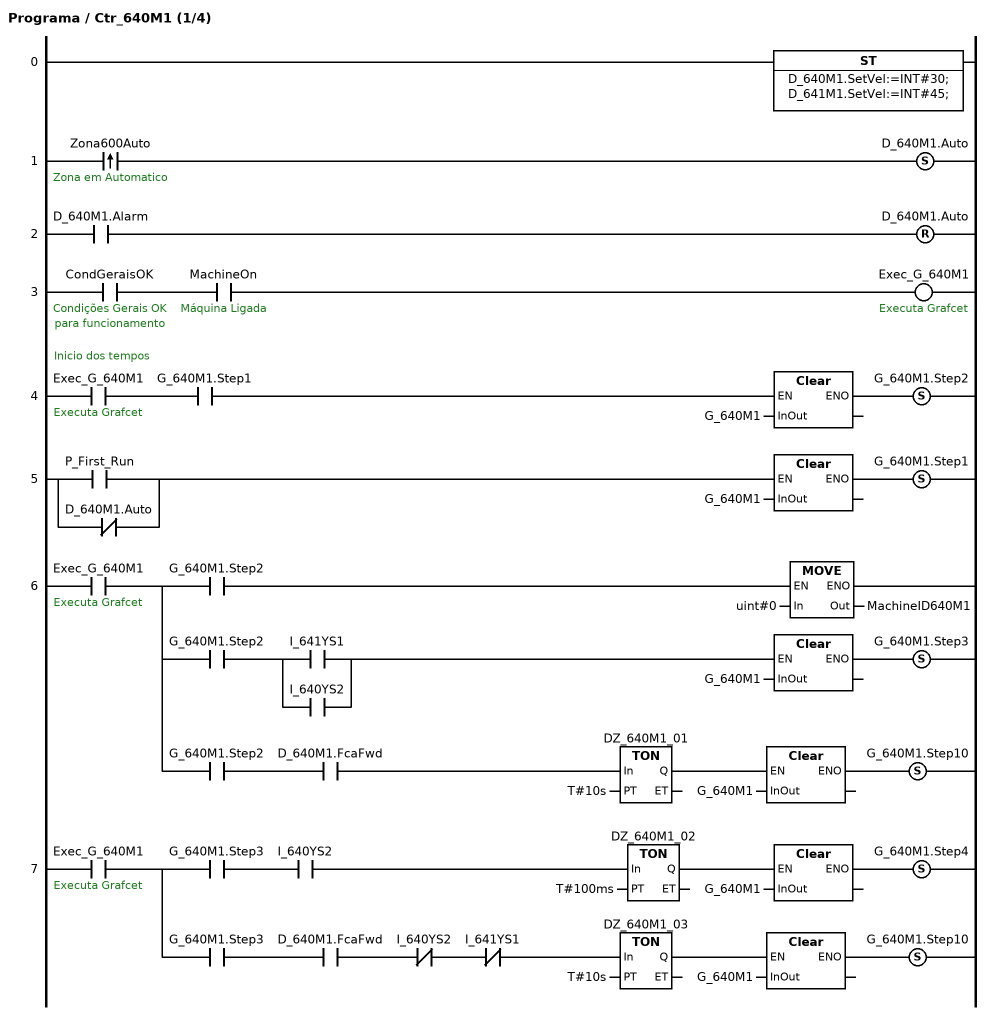
(* [picture p144: Programa / Ctr_640M1, rungs 0-7] *)
(* Rung 0 *)
D_640M1.SetVel:=INT#30;
D_641M1.SetVel:=INT#45;
(* Rung 1 *)
_e291(CLK := Zona600Auto);
IF _e291.Q THEN D_640M1.Auto := TRUE; END_IF;
(* Rung 2 *)
IF D_640M1.Alarm THEN D_640M1.Auto := FALSE; END_IF;
(* Rung 3 *)
Exec_G_640M1 := CondGeraisOK AND MachineOn;
(* Rung 4: Inicio dos tempos *)
_p292 := Exec_G_640M1 AND G_640M1.Step1;
IF _p292 THEN
    Clear(InOut := G_640M1);
    G_640M1.Step2 := TRUE;
END_IF;
(* Rung 5 *)
IF P_First_Run OR NOT D_640M1.Auto THEN
    Clear(InOut := G_640M1);
    G_640M1.Step1 := TRUE;
END_IF;
(* Rung 6 *)
IF Exec_G_640M1 AND G_640M1.Step2 THEN MachineID640M1 := uint#0; END_IF;
_p293 := Exec_G_640M1 AND G_640M1.Step2 AND (I_641YS1 OR I_640YS2);
IF _p293 THEN
    Clear(InOut := G_640M1);
    G_640M1.Step3 := TRUE;
END_IF;
DZ_640M1_01(In := Exec_G_640M1 AND G_640M1.Step2 AND D_640M1.FcaFwd, PT := T#10s);
IF DZ_640M1_01.Q THEN
    Clear(InOut := G_640M1);
    G_640M1.Step10 := TRUE;
END_IF;
(* Rung 7 *)
DZ_640M1_02(In := Exec_G_640M1 AND G_640M1.Step3 AND I_640YS2, PT := T#100ms);
IF DZ_640M1_02.Q THEN
    Clear(InOut := G_640M1);
    G_640M1.Step4 := TRUE;
END_IF;
DZ_640M1_03(In := Exec_G_640M1 AND G_640M1.Step3 AND D_640M1.FcaFwd AND NOT I_640YS2 AND NOT I_641YS1, PT := T#10s);
IF DZ_640M1_03.Q THEN
    Clear(InOut := G_640M1);
    G_640M1.Step10 := TRUE;
END_IF;

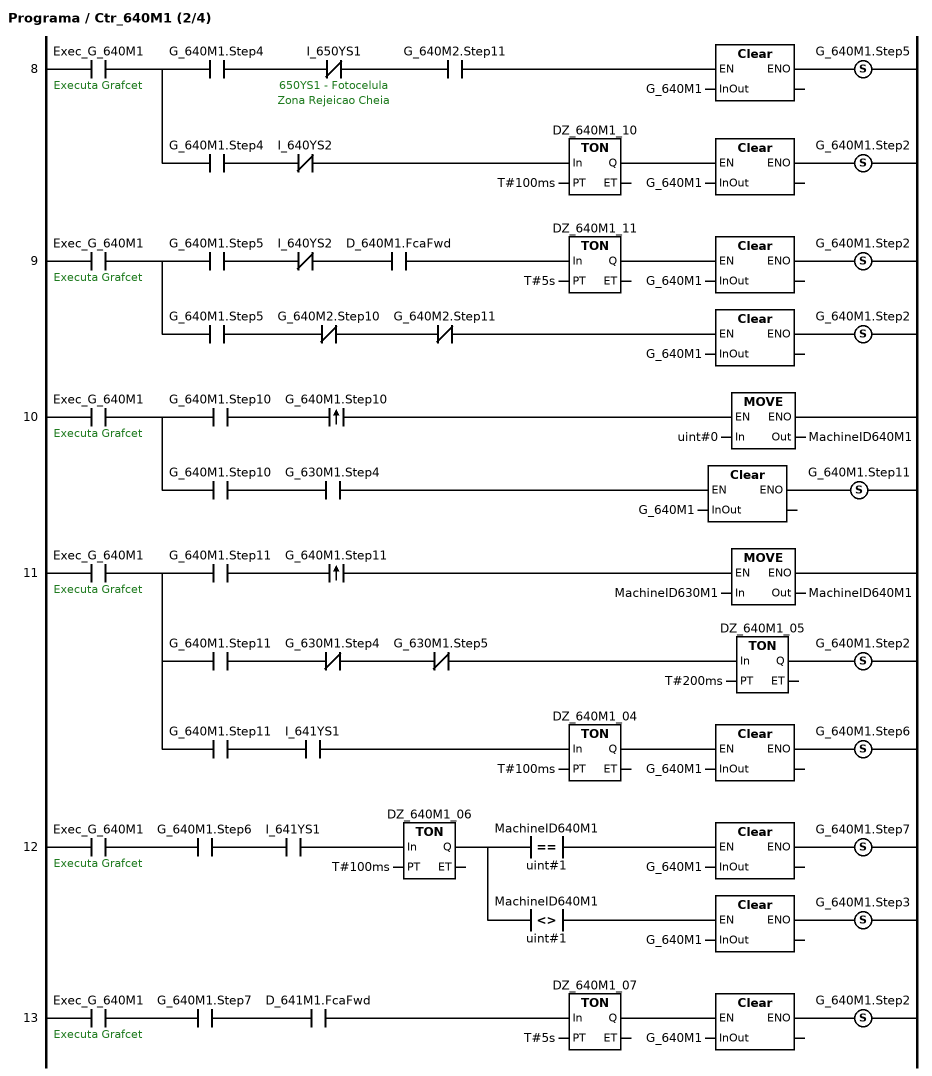
(* Rung 8 *)
_p294 := Exec_G_640M1 AND G_640M1.Step4 AND NOT I_650YS1 AND G_640M2.Step11;
IF _p294 THEN
    Clear(InOut := G_640M1);
    G_640M1.Step5 := TRUE;
END_IF;
DZ_640M1_10(In := Exec_G_640M1 AND G_640M1.Step4 AND NOT I_640YS2, PT := T#100ms);
IF DZ_640M1_10.Q THEN
    Clear(InOut := G_640M1);
    G_640M1.Step2 := TRUE;
END_IF;
(* Rung 9 *)
DZ_640M1_11(In := Exec_G_640M1 AND G_640M1.Step5 AND NOT I_640YS2 AND D_640M1.FcaFwd, PT := T#5s);
IF DZ_640M1_11.Q THEN
    Clear(InOut := G_640M1);
    G_640M1.Step2 := TRUE;
END_IF;
_p295 := Exec_G_640M1 AND G_640M1.Step5 AND NOT G_640M2.Step10 AND NOT G_640M2.Step11;
IF _p295 THEN
    Clear(InOut := G_640M1);
    G_640M1.Step2 := TRUE;
END_IF;
(* Rung 10 *)
_e296(CLK := G_640M1.Step10);
IF Exec_G_640M1 AND G_640M1.Step10 AND _e296.Q THEN MachineID640M1 := uint#0; END_IF;
_p297 := Exec_G_640M1 AND G_640M1.Step10 AND G_630M1.Step4;
IF _p297 THEN
    Clear(InOut := G_640M1);
    G_640M1.Step11 := TRUE;
END_IF;
(* Rung 11 *)
_e298(CLK := G_640M1.Step11);
IF Exec_G_640M1 AND G_640M1.Step11 AND _e298.Q THEN MachineID640M1 := MachineID630M1; END_IF;
DZ_640M1_05(In := Exec_G_640M1 AND G_640M1.Step11 AND NOT G_630M1.Step4 AND NOT G_630M1.Step5, PT := T#200ms);
IF DZ_640M1_05.Q THEN G_640M1.Step2 := TRUE; END_IF;
DZ_640M1_04(In := Exec_G_640M1 AND G_640M1.Step11 AND I_641YS1, PT := T#100ms);
IF DZ_640M1_04.Q THEN
    Clear(InOut := G_640M1);
    G_640M1.Step6 := TRUE;
END_IF;
(* Rung 12 *)
DZ_640M1_06(In := Exec_G_640M1 AND G_640M1.Step6 AND I_641YS1, PT := T#100ms);
IF DZ_640M1_06.Q AND (MachineID640M1 = uint#1) THEN
    Clear(InOut := G_640M1);
    G_640M1.Step7 := TRUE;
END_IF;
IF DZ_640M1_06.Q AND (MachineID640M1 <> uint#1) THEN
    Clear(InOut := G_640M1);
    G_640M1.Step3 := TRUE;
END_IF;
(* Rung 13 *)
DZ_640M1_07(In := Exec_G_640M1 AND G_640M1.Step7 AND D_641M1.FcaFwd, PT := T#5s);
IF DZ_640M1_07.Q THEN
    Clear(InOut := G_640M1);
    G_640M1.Step2 := TRUE;
END_IF;

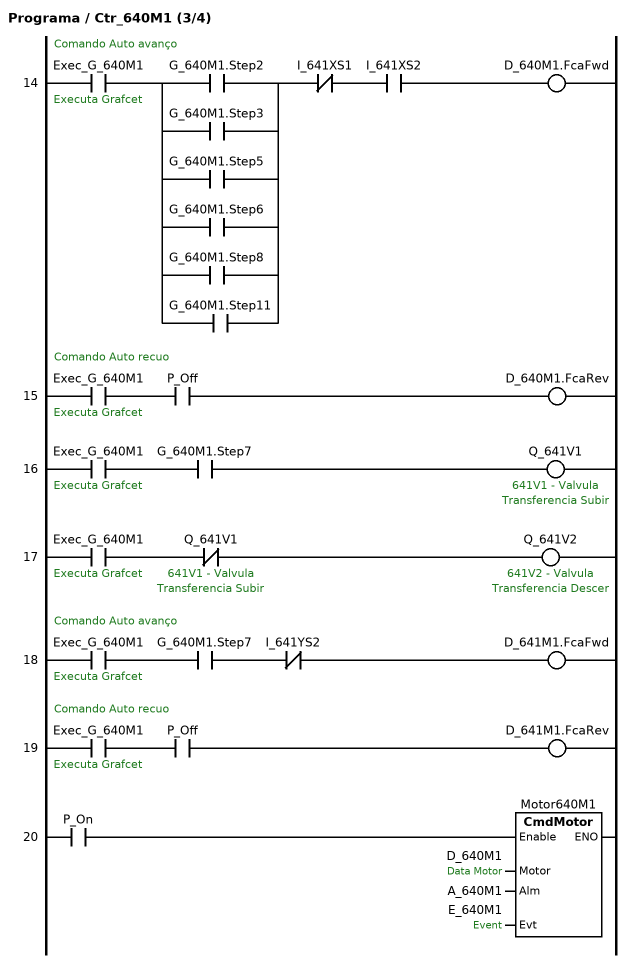
(* Rung 14: Comando Auto avanço *)
D_640M1.FcaFwd := Exec_G_640M1 AND (G_640M1.Step2 OR G_640M1.Step3 OR G_640M1.Step5 OR G_640M1.Step6 OR G_640M1.Step8 OR G_640M1.Step11) AND NOT I_641XS1 AND I_641XS2;
(* Rung 15: Comando Auto recuo *)
D_640M1.FcaRev := Exec_G_640M1 AND P_Off;
(* Rung 16 *)
Q_641V1 := Exec_G_640M1 AND G_640M1.Step7;
(* Rung 17 *)
Q_641V2 := Exec_G_640M1 AND NOT Q_641V1;
(* Rung 18: Comando Auto avanço *)
D_641M1.FcaFwd := Exec_G_640M1 AND G_640M1.Step7 AND NOT I_641YS2;
(* Rung 19: Comando Auto recuo *)
D_641M1.FcaRev := Exec_G_640M1 AND P_Off;
(* Rung 20 *)
Motor640M1(Enable := P_On, Motor := D_640M1, Alm := A_640M1, Evt := E_640M1);

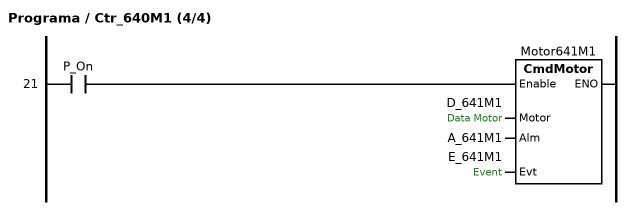
(* Rung 21 *)
Motor641M1(Enable := P_On, Motor := D_641M1, Alm := A_641M1, Evt := E_641M1);

(* Section Ctr_640M2: ladder, written here as Structured Text *)

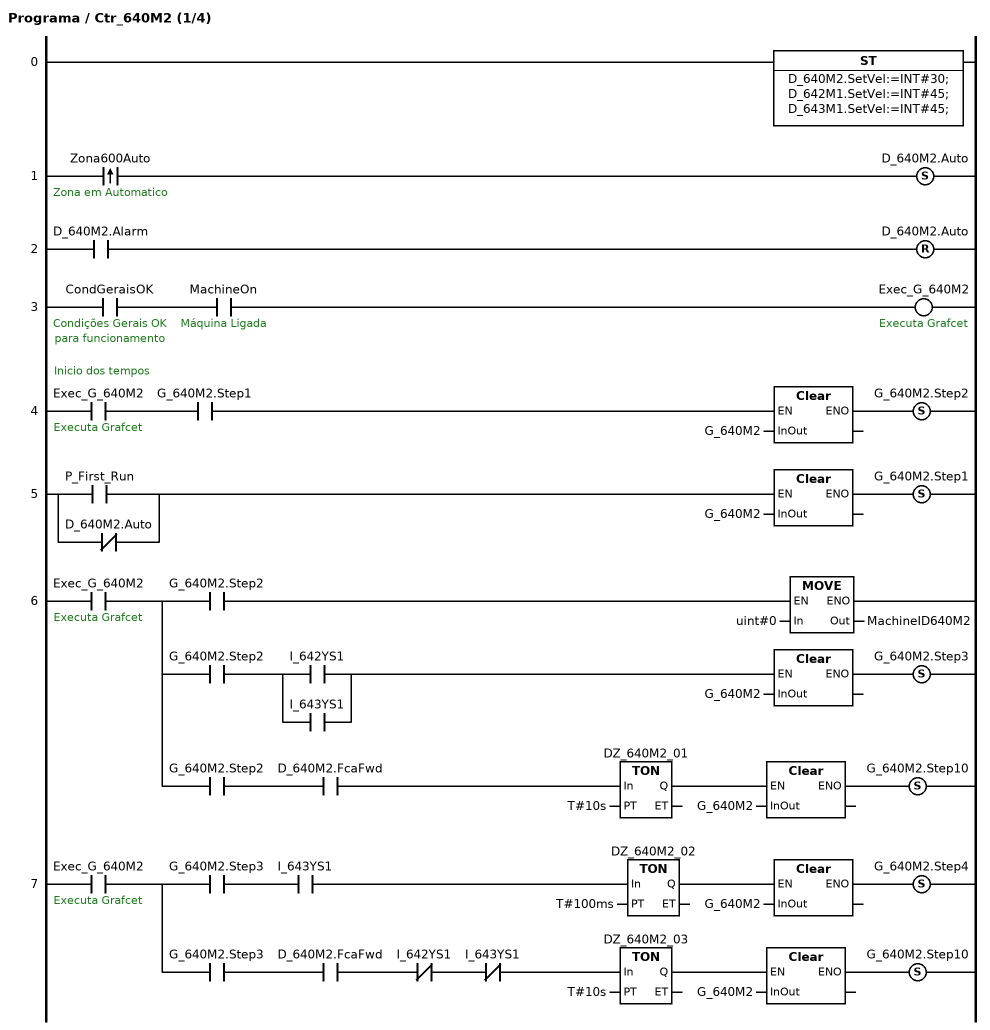
(* Rung 0 *)
D_640M2.SetVel:=INT#30;
D_642M1.SetVel:=INT#45;
D_643M1.SetVel:=INT#45;
(* Rung 1 *)
_e299(CLK := Zona600Auto);
IF _e299.Q THEN D_640M2.Auto := TRUE; END_IF;
(* Rung 2 *)
IF D_640M2.Alarm THEN D_640M2.Auto := FALSE; END_IF;
(* Rung 3 *)
Exec_G_640M2 := CondGeraisOK AND MachineOn;
(* Rung 4: Inicio dos tempos *)
_p300 := Exec_G_640M2 AND G_640M2.Step1;
IF _p300 THEN
    Clear(InOut := G_640M2);
    G_640M2.Step2 := TRUE;
END_IF;
(* Rung 5 *)
IF P_First_Run OR NOT D_640M2.Auto THEN
    Clear(InOut := G_640M2);
    G_640M2.Step1 := TRUE;
END_IF;
(* Rung 6 *)
IF Exec_G_640M2 AND G_640M2.Step2 THEN MachineID640M2 := uint#0; END_IF;
_p301 := Exec_G_640M2 AND G_640M2.Step2 AND (I_642YS1 OR I_643YS1);
IF _p301 THEN
    Clear(InOut := G_640M2);
    G_640M2.Step3 := TRUE;
END_IF;
DZ_640M2_01(In := Exec_G_640M2 AND G_640M2.Step2 AND D_640M2.FcaFwd, PT := T#10s);
IF DZ_640M2_01.Q THEN
    Clear(InOut := G_640M2);
    G_640M2.Step10 := TRUE;
END_IF;
(* Rung 7 *)
DZ_640M2_02(In := Exec_G_640M2 AND G_640M2.Step3 AND I_643YS1, PT := T#100ms);
IF DZ_640M2_02.Q THEN
    Clear(InOut := G_640M2);
    G_640M2.Step4 := TRUE;
END_IF;
DZ_640M2_03(In := Exec_G_640M2 AND G_640M2.Step3 AND D_640M2.FcaFwd AND NOT I_642YS1 AND NOT I_643YS1, PT := T#10s);
IF DZ_640M2_03.Q THEN
    Clear(InOut := G_640M2);
    G_640M2.Step10 := TRUE;
END_IF;

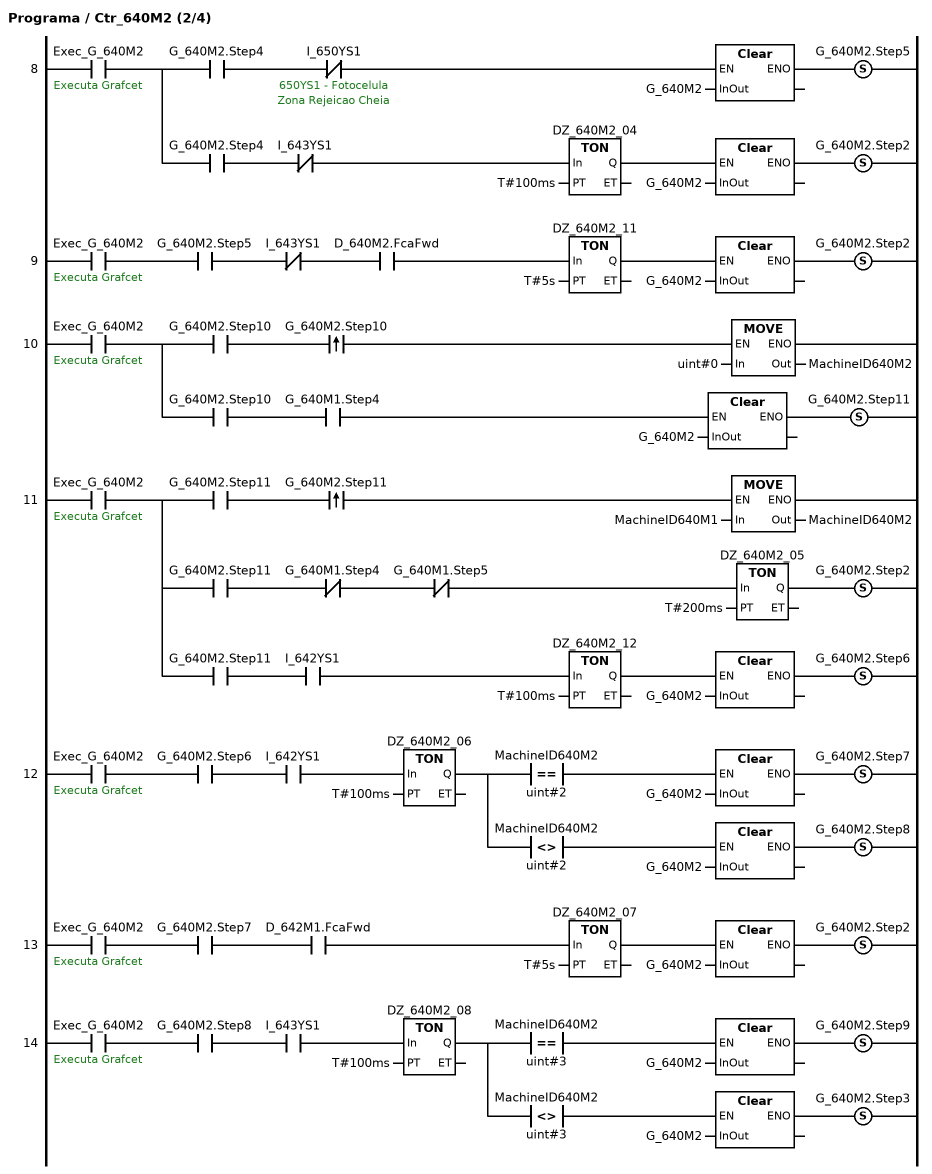
(* Rung 8 *)
_p302 := Exec_G_640M2 AND G_640M2.Step4 AND NOT I_650YS1;
IF _p302 THEN
    Clear(InOut := G_640M2);
    G_640M2.Step5 := TRUE;
END_IF;
DZ_640M2_04(In := Exec_G_640M2 AND G_640M2.Step4 AND NOT I_643YS1, PT := T#100ms);
IF DZ_640M2_04.Q THEN
    Clear(InOut := G_640M2);
    G_640M2.Step2 := TRUE;
END_IF;
(* Rung 9 *)
DZ_640M2_11(In := Exec_G_640M2 AND G_640M2.Step5 AND NOT I_643YS1 AND D_640M2.FcaFwd, PT := T#5s);
IF DZ_640M2_11.Q THEN
    Clear(InOut := G_640M2);
    G_640M2.Step2 := TRUE;
END_IF;
(* Rung 10 *)
_e303(CLK := G_640M2.Step10);
IF Exec_G_640M2 AND G_640M2.Step10 AND _e303.Q THEN MachineID640M2 := uint#0; END_IF;
_p304 := Exec_G_640M2 AND G_640M2.Step10 AND G_640M1.Step4;
IF _p304 THEN
    Clear(InOut := G_640M2);
    G_640M2.Step11 := TRUE;
END_IF;
(* Rung 11 *)
_e305(CLK := G_640M2.Step11);
IF Exec_G_640M2 AND G_640M2.Step11 AND _e305.Q THEN MachineID640M2 := MachineID640M1; END_IF;
DZ_640M2_05(In := Exec_G_640M2 AND G_640M2.Step11 AND NOT G_640M1.Step4 AND NOT G_640M1.Step5, PT := T#200ms);
IF DZ_640M2_05.Q THEN G_640M2.Step2 := TRUE; END_IF;
DZ_640M2_12(In := Exec_G_640M2 AND G_640M2.Step11 AND I_642YS1, PT := T#100ms);
IF DZ_640M2_12.Q THEN
    Clear(InOut := G_640M2);
    G_640M2.Step6 := TRUE;
END_IF;
(* Rung 12 *)
DZ_640M2_06(In := Exec_G_640M2 AND G_640M2.Step6 AND I_642YS1, PT := T#100ms);
IF DZ_640M2_06.Q AND (MachineID640M2 = uint#2) THEN
    Clear(InOut := G_640M2);
    G_640M2.Step7 := TRUE;
END_IF;
IF DZ_640M2_06.Q AND (MachineID640M2 <> uint#2) THEN
    Clear(InOut := G_640M2);
    G_640M2.Step8 := TRUE;
END_IF;
(* Rung 13 *)
DZ_640M2_07(In := Exec_G_640M2 AND G_640M2.Step7 AND D_642M1.FcaFwd, PT := T#5s);
IF DZ_640M2_07.Q THEN
    Clear(InOut := G_640M2);
    G_640M2.Step2 := TRUE;
END_IF;
(* Rung 14 *)
DZ_640M2_08(In := Exec_G_640M2 AND G_640M2.Step8 AND I_643YS1, PT := T#100ms);
IF DZ_640M2_08.Q AND (MachineID640M2 = uint#3) THEN
    Clear(InOut := G_640M2);
    G_640M2.Step9 := TRUE;
END_IF;
IF DZ_640M2_08.Q AND (MachineID640M2 <> uint#3) THEN
    Clear(InOut := G_640M2);
    G_640M2.Step3 := TRUE;
END_IF;

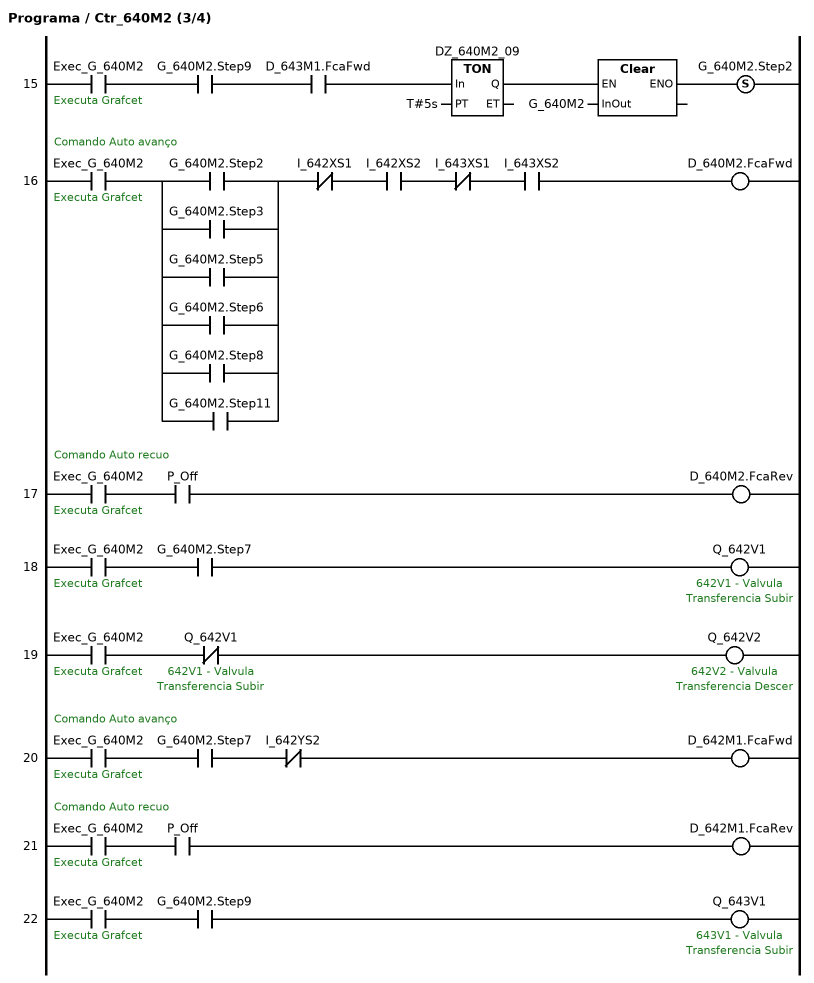
(* Rung 15 *)
DZ_640M2_09(In := Exec_G_640M2 AND G_640M2.Step9 AND D_643M1.FcaFwd, PT := T#5s);
IF DZ_640M2_09.Q THEN
    Clear(InOut := G_640M2);
    G_640M2.Step2 := TRUE;
END_IF;
(* Rung 16: Comando Auto avanço *)
D_640M2.FcaFwd := Exec_G_640M2 AND (G_640M2.Step2 OR G_640M2.Step3 OR G_640M2.Step5 OR G_640M2.Step6 OR G_640M2.Step8 OR G_640M2.Step11) AND NOT I_642XS1 AND I_642XS2 AND NOT I_643XS1 AND I_643XS2;
(* Rung 17: Comando Auto recuo *)
D_640M2.FcaRev := Exec_G_640M2 AND P_Off;
(* Rung 18 *)
Q_642V1 := Exec_G_640M2 AND G_640M2.Step7;
(* Rung 19 *)
Q_642V2 := Exec_G_640M2 AND NOT Q_642V1;
(* Rung 20: Comando Auto avanço *)
D_642M1.FcaFwd := Exec_G_640M2 AND G_640M2.Step7 AND NOT I_642YS2;
(* Rung 21: Comando Auto recuo *)
D_642M1.FcaRev := Exec_G_640M2 AND P_Off;
(* Rung 22 *)
Q_643V1 := Exec_G_640M2 AND G_640M2.Step9;

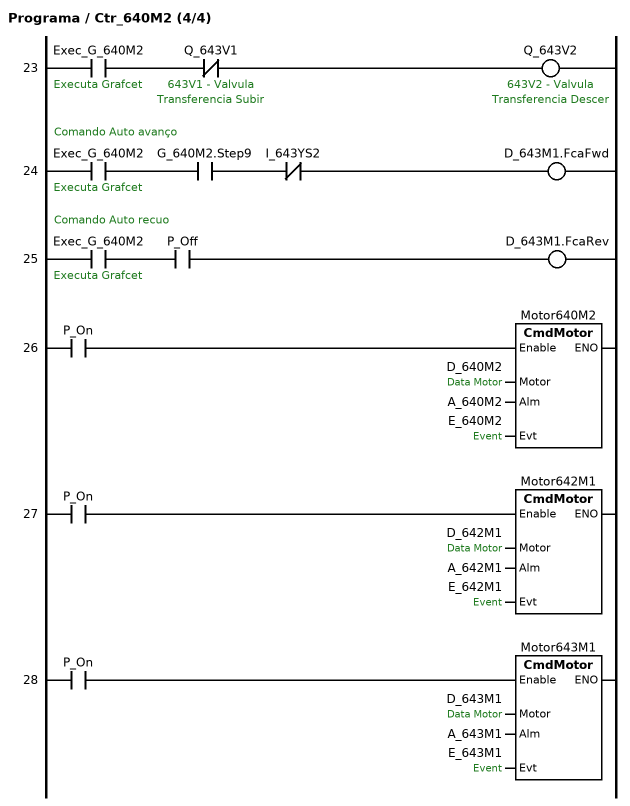
(* Rung 23 *)
Q_643V2 := Exec_G_640M2 AND NOT Q_643V1;
(* Rung 24: Comando Auto avanço *)
D_643M1.FcaFwd := Exec_G_640M2 AND G_640M2.Step9 AND NOT I_643YS2;
(* Rung 25: Comando Auto recuo *)
D_643M1.FcaRev := Exec_G_640M2 AND P_Off;
(* Rung 26 *)
Motor640M2(Enable := P_On, Motor := D_640M2, Alm := A_640M2, Evt := E_640M2);
(* Rung 27 *)
Motor642M1(Enable := P_On, Motor := D_642M1, Alm := A_642M1, Evt := E_642M1);
(* Rung 28 *)
Motor643M1(Enable := P_On, Motor := D_643M1, Alm := A_643M1, Evt := E_643M1);

(* Section Ctr_020A1_G9SP: ladder, written here as Structured Text *)

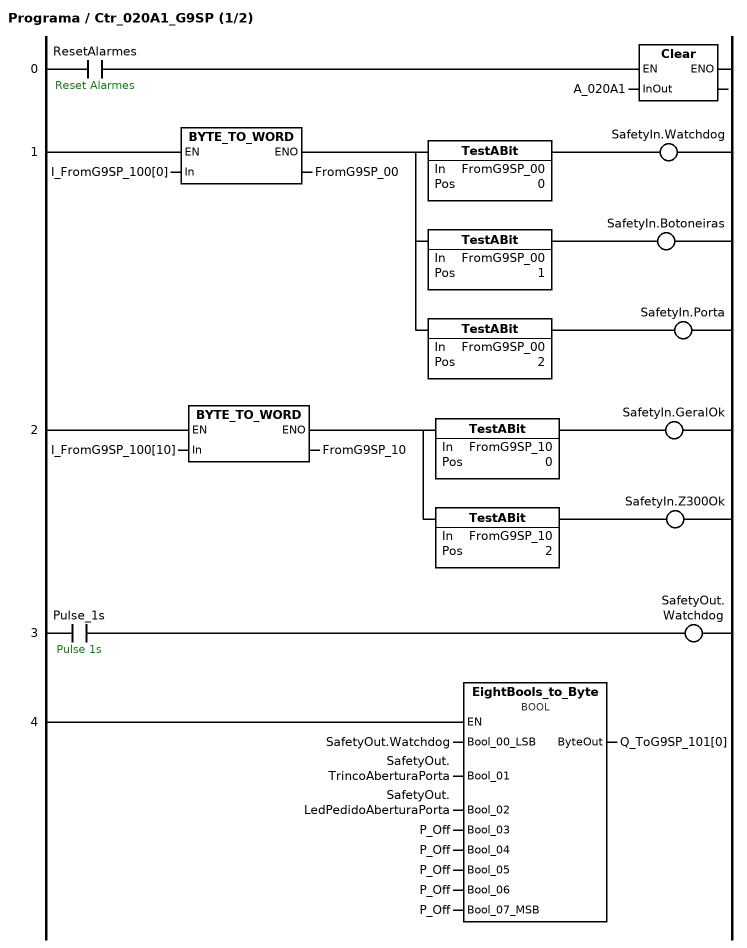
(* Rung 0 *)
IF ResetAlarmes THEN Clear(InOut := A_020A1); END_IF;
(* Rung 1 *)
FromG9SP_00 := BYTE_TO_WORD(In := I_FromG9SP_100[0]);
SafetyIn.Watchdog := TestABit(In := FromG9SP_00, Pos := 0);
SafetyIn.Botoneiras := TestABit(In := FromG9SP_00, Pos := 1);
SafetyIn.Porta := TestABit(In := FromG9SP_00, Pos := 2);
(* Rung 2 *)
FromG9SP_10 := BYTE_TO_WORD(In := I_FromG9SP_100[10]);
SafetyIn.GeralOk := TestABit(In := FromG9SP_10, Pos := 0);
SafetyIn.Z300Ok := TestABit(In := FromG9SP_10, Pos := 2);
(* Rung 3 *)
SafetyOut.Watchdog := Pulse_1s;
(* Rung 4 *)
_t306 := EightBools_to_Byte(Bool_00_LSB := SafetyOut.Watchdog, Bool_01 := SafetyOut.TrincoAberturaPorta, Bool_02 := SafetyOut.LedPedidoAberturaPorta, Bool_03 := P_Off, Bool_04 := P_Off, Bool_05 := P_Off, Bool_06 := P_Off, Bool_07_MSB := P_Off, ByteOut => Q_ToG9SP_101[0]);

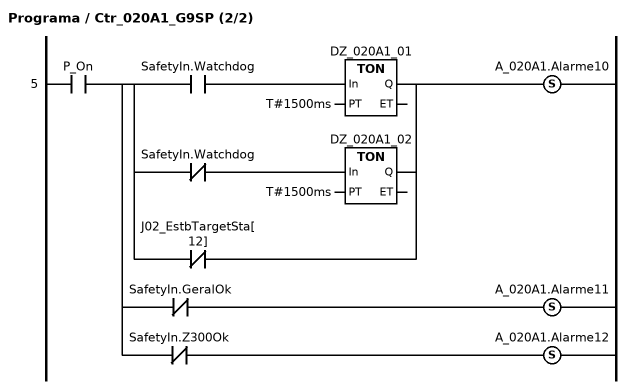
(* Rung 5 *)
DZ_020A1_01(In := P_On AND SafetyIn.Watchdog, PT := T#1500ms);
DZ_020A1_02(In := P_On AND NOT SafetyIn.Watchdog, PT := T#1500ms);
IF DZ_020A1_01.Q OR DZ_020A1_02.Q OR (P_On AND NOT J02_EstbTargetSta[12]) THEN
    A_020A1.Alarme10 := TRUE;
END_IF;
IF P_On AND NOT SafetyIn.GeralOk THEN A_020A1.Alarme11 := TRUE; END_IF;
IF P_On AND NOT SafetyIn.Z300Ok THEN A_020A1.Alarme12 := TRUE; END_IF;

(* Section Ctr_ICM500_600: ladder, written here as Structured Text *)

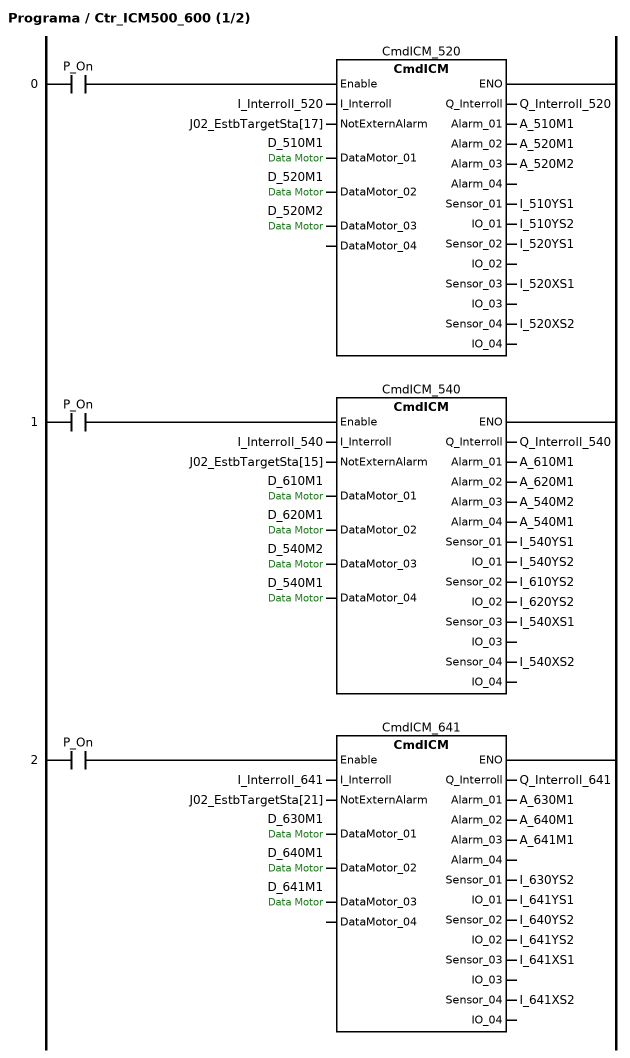
(* Rung 0 *)
CmdICM_520(Enable := P_On, I_Interroll := I_Interroll_520, NotExternAlarm := J02_EstbTargetSta[17], DataMotor_01 := D_510M1, DataMotor_02 := D_520M1, DataMotor_03 := D_520M2, Q_Interroll => Q_Interroll_520, Alarm_01 => A_510M1, Alarm_02 => A_520M1, Alarm_03 => A_520M2, Sensor_01 => I_510YS1, IO_01 => I_510YS2, Sensor_02 => I_520YS1, Sensor_03 => I_520XS1, Sensor_04 => I_520XS2);
(* Rung 1 *)
CmdICM_540(Enable := P_On, I_Interroll := I_Interroll_540, NotExternAlarm := J02_EstbTargetSta[15], DataMotor_01 := D_610M1, DataMotor_02 := D_620M1, DataMotor_03 := D_540M2, DataMotor_04 := D_540M1, Q_Interroll => Q_Interroll_540, Alarm_01 => A_610M1, Alarm_02 => A_620M1, Alarm_03 => A_540M2, Alarm_04 => A_540M1, Sensor_01 => I_540YS1, IO_01 => I_540YS2, Sensor_02 => I_610YS2, IO_02 => I_620YS2, Sensor_03 => I_540XS1, Sensor_04 => I_540XS2);
(* Rung 2 *)
CmdICM_641(Enable := P_On, I_Interroll := I_Interroll_641, NotExternAlarm := J02_EstbTargetSta[21], DataMotor_01 := D_630M1, DataMotor_02 := D_640M1, DataMotor_03 := D_641M1, Q_Interroll => Q_Interroll_641, Alarm_01 => A_630M1, Alarm_02 => A_640M1, Alarm_03 => A_641M1, Sensor_01 => I_630YS2, IO_01 => I_641YS1, Sensor_02 => I_640YS2, IO_02 => I_641YS2, Sensor_03 => I_641XS1, Sensor_04 => I_641XS2);

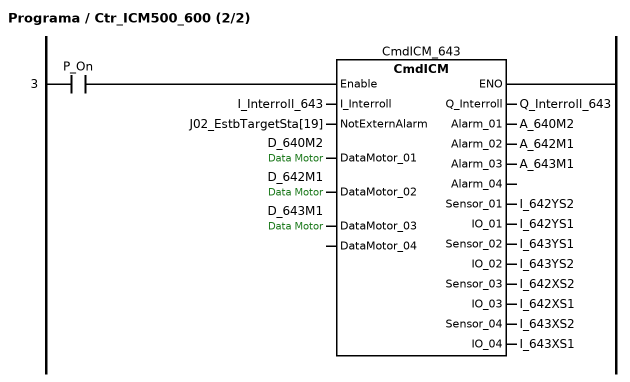
(* Rung 3 *)
CmdICM_643(Enable := P_On, I_Interroll := I_Interroll_643, NotExternAlarm := J02_EstbTargetSta[19], DataMotor_01 := D_640M2, DataMotor_02 := D_642M1, DataMotor_03 := D_643M1, Q_Interroll => Q_Interroll_643, Alarm_01 => A_640M2, Alarm_02 => A_642M1, Alarm_03 => A_643M1, Sensor_01 => I_642YS2, IO_01 => I_642YS1, Sensor_02 => I_643YS1, IO_02 => I_643YS2, Sensor_03 => I_642XS2, IO_03 => I_642XS1, Sensor_04 => I_643XS2, IO_04 => I_643XS1);
END_PROGRAM

FUNCTION Int_to_BitArray16 : BOOL
VAR
    MyInt : UINT;
END_VAR
VAR_INPUT
    Input_Int : INT;
END_VAR
VAR_OUTPUT
    BitArray16_out : array[0..15] of bool;
END_VAR
MyInt:=real_to_int(Input_Int);
//MyInt:=1025;
IF (MyInt/(2**15))>=1 THEN BitArray16_out[15]:=true; MyInt:=MyInt-(2**15); ELSE  BitArray16_out[15]:=false; END_IF;
IF (MyInt/(2**14))>=1 THEN BitArray16_out[14]:=true; MyInt:=MyInt-(2**14); ELSE  BitArray16_out[14]:=false; END_IF;
IF (MyInt/(2**13))>=1 THEN BitArray16_out[13]:=true; MyInt:=MyInt-(2**13); ELSE  BitArray16_out[13]:=false; END_IF;
IF (MyInt/(2**12))>=1 THEN BitArray16_out[12]:=true; MyInt:=MyInt-(2**12); ELSE  BitArray16_out[12]:=false; END_IF;
IF (MyInt/(2**11))>=1 THEN BitArray16_out[11]:=true; MyInt:=MyInt-(2**11); ELSE  BitArray16_out[11]:=false; END_IF;
IF (MyInt/(2**10))>=1 THEN BitArray16_out[10]:=true; MyInt:=MyInt-(2**10); ELSE  BitArray16_out[10]:=false; END_IF;
IF (MyInt/(2**09))>=1 THEN BitArray16_out[09]:=true; MyInt:=MyInt-(2**09); ELSE  BitArray16_out[09]:=false; END_IF;
IF (MyInt/(2**08))>=1 THEN BitArray16_out[08]:=true; MyInt:=MyInt-(2**08); ELSE  BitArray16_out[08]:=false; END_IF;
IF (MyInt/(2**07))>=1 THEN BitArray16_out[07]:=true; MyInt:=MyInt-(2**07); ELSE  BitArray16_out[07]:=false; END_IF;
IF (MyInt/(2**06))>=1 THEN BitArray16_out[06]:=true; MyInt:=MyInt-(2**06); ELSE  BitArray16_out[06]:=false; END_IF;
IF (MyInt/(2**05))>=1 THEN BitArray16_out[05]:=true; MyInt:=MyInt-(2**05); ELSE  BitArray16_out[05]:=false; END_IF;
IF (MyInt/(2**04))>=1 THEN BitArray16_out[04]:=true; MyInt:=MyInt-(2**04); ELSE  BitArray16_out[04]:=false; END_IF;
IF (MyInt/(2**03))>=1 THEN BitArray16_out[03]:=true; MyInt:=MyInt-(2**03); ELSE  BitArray16_out[03]:=false; END_IF;
IF (MyInt/(2**02))>=1 THEN BitArray16_out[02]:=true; MyInt:=MyInt-(2**02); ELSE  BitArray16_out[02]:=false; END_IF;
IF (MyInt/(2**01))>=1 THEN BitArray16_out[01]:=true; MyInt:=MyInt-(2**01); ELSE  BitArray16_out[01]:=false; END_IF;
IF (MyInt/(2**00))>=1 THEN BitArray16_out[00]:=true; MyInt:=MyInt-(2**00); ELSE  BitArray16_out[00]:=false; END_IF;
END_FUNCTION

FUNCTION BitArray16_to_UInt : UINT
VAR
    UIntOut : UINT;
END_VAR
VAR_INPUT
    ArrayIn : array[0..15] of bool;
END_VAR
UIntOut:=0;
If ArrayIn[0] then UIntOut :=UIntOut+1*(2**0); END_IF;
If ArrayIn[1] then UIntOut :=UIntOut+1*(2**1); END_IF;
If ArrayIn[2] then UIntOut :=UIntOut+1*(2**2); END_IF;
If ArrayIn[3] then UIntOut :=UIntOut+1*(2**3); END_IF;
If ArrayIn[4] then UIntOut :=UIntOut+1*(2**4); END_IF;
If ArrayIn[5] then UIntOut :=UIntOut+1*(2**5); END_IF;
If ArrayIn[6] then UIntOut :=UIntOut+1*(2**6); END_IF;
If ArrayIn[7] then UIntOut :=UIntOut+1*(2**7); END_IF;
If ArrayIn[8] then UIntOut :=UIntOut+1*(2**8); END_IF;
If ArrayIn[9] then UIntOut :=UIntOut+1*(2**9); END_IF;
If ArrayIn[10] then UIntOut :=UIntOut+1*(2**10); END_IF;
If ArrayIn[11] then UIntOut :=UIntOut+1*(2**11); END_IF;
If ArrayIn[12] then UIntOut :=UIntOut+1*(2**12); END_IF;
If ArrayIn[13] then UIntOut :=UIntOut+1*(2**13); END_IF;
If ArrayIn[14] then UIntOut :=UIntOut+1*(2**14); END_IF;
If ArrayIn[15] then UIntOut :=UIntOut+1*(2**15); END_IF;
BitArray16_to_UInt:=UIntOut;
END_FUNCTION

FUNCTION IntAscii2Char : BOOL
VAR_INPUT
    HexIntAsciiValue : INT;
END_VAR
VAR_OUTPUT
    OutChar : String[2];
END_VAR
CASE HexIntAsciiValue OF
	16#30: OutChar:='0';
	16#31: OutChar:='1';
	16#32: OutChar:='2';
	16#33: OutChar:='3';
	16#34: OutChar:='4';
	16#35: OutChar:='5';
	16#36: OutChar:='6';
	16#37: OutChar:='7';
	16#38: OutChar:='8';
	16#39: OutChar:='9';
	16#3B: OutChar:=';';
	16#41: OutChar:='A';
	16#42: OutChar:='B';
	16#43: OutChar:='C';
	16#44: OutChar:='D';
	16#45: OutChar:='E';
	16#46: OutChar:='F';
	16#47: OutChar:='G';
	16#48: OutChar:='H';
	16#49: OutChar:='I';
	16#4A: OutChar:='J';
	16#4B: OutChar:='K';
	16#4C: OutChar:='L';
	16#4D: OutChar:='M';
	16#4E: OutChar:='N';
	16#4F: OutChar:='O';
	16#50: OutChar:='P';
	16#51: OutChar:='Q';
	16#52: OutChar:='R';
	16#53: OutChar:='S';
	16#54: OutChar:='T';
	16#55: OutChar:='U';
	16#56: OutChar:='V';
	16#57: OutChar:='W';
	16#58: OutChar:='X';
	16#59: OutChar:='Y';
	16#5A: OutChar:='Z';
ELSE
OutChar:='-';
END_CASE;	
		
END_FUNCTION

FUNCTION EightBools_to_Byte : BOOL
VAR_INPUT
    Bool_00_LSB : BOOL;
    Bool_01 : BOOL;
    Bool_02 : BOOL;
    Bool_03 : BOOL;
    Bool_04 : BOOL;
    Bool_05 : BOOL;
    Bool_06 : BOOL;
    Bool_07_MSB : BOOL;
END_VAR
VAR_OUTPUT
    ByteOut : BYTE;
END_VAR
(* ladder, written here as Structured Text *)

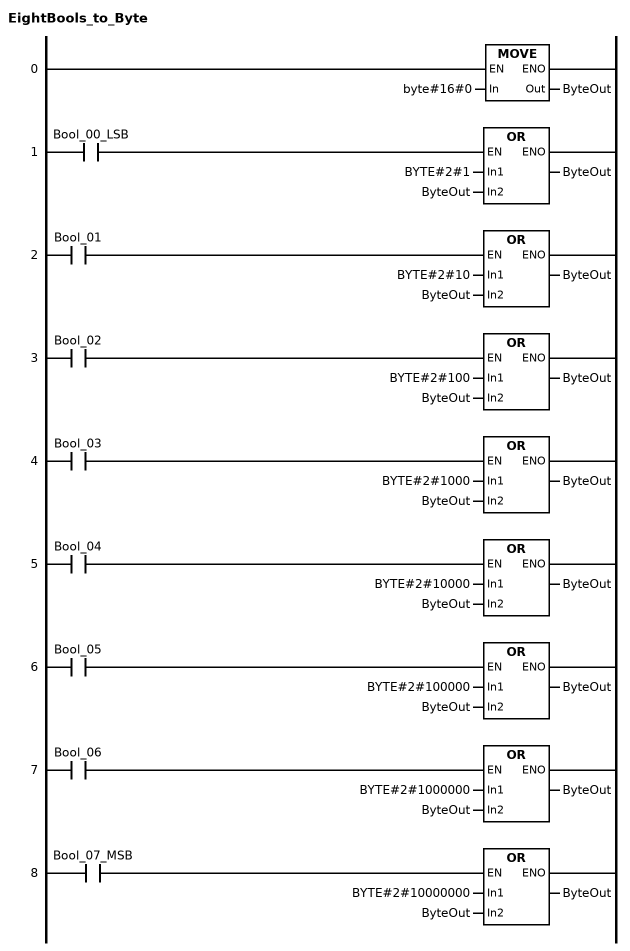
(* Rung 0 *)
ByteOut := byte#16#0;
(* Rung 1 *)
IF Bool_00_LSB THEN ByteOut := BYTE#2#1 OR ByteOut; END_IF;
(* Rung 2 *)
IF Bool_01 THEN ByteOut := BYTE#2#10 OR ByteOut; END_IF;
(* Rung 3 *)
IF Bool_02 THEN ByteOut := BYTE#2#100 OR ByteOut; END_IF;
(* Rung 4 *)
IF Bool_03 THEN ByteOut := BYTE#2#1000 OR ByteOut; END_IF;
(* Rung 5 *)
IF Bool_04 THEN ByteOut := BYTE#2#10000 OR ByteOut; END_IF;
(* Rung 6 *)
IF Bool_05 THEN ByteOut := BYTE#2#100000 OR ByteOut; END_IF;
(* Rung 7 *)
IF Bool_06 THEN ByteOut := BYTE#2#1000000 OR ByteOut; END_IF;
(* Rung 8 *)
IF Bool_07_MSB THEN ByteOut := BYTE#2#10000000 OR ByteOut; END_IF;
END_FUNCTION

FUNCTION_BLOCK CmdLenzeI550
VAR
    ReadyToSwitchOn : BOOL;
    SwitchedOn : BOOL;
    OperationEnabled : BOOL;
    FaultActive : BOOL;
    VoltageEnabled : BOOL;
    In_QuickStop : BOOL;
    SwitchOnDisabled : BOOL;
    WarningActive : BOOL;
    DeactivateRPDOs : BOOL;
    Remote : BOOL;
    TargetReached : BOOL;
    InternalLimitActive : BOOL;
    OperationModeActive : BOOL;
    FollowingError : BOOL;
    HoldingBrakeReleased : BOOL;
    SafeTorqueOffNotActive : BOOL;
    Status16 : WORD;
    MyArray : array[0..15] of bool;
    SwitchOn : BOOL;
    EnableVoltage : BOOL;
    Out_QuickStop : BOOL;
    EnableOperation : BOOL;
END_VAR
VAR_IN_OUT
    Motor : DataMotor;  (* Data *)
    Alm : AlarmeGeralEquipamento;  (* Alarme *)
    Evt : Event;  (* Event *)
END_VAR
VAR_INPUT
    Enable : BOOL;
    StatusWord : UINT;
END_VAR
VAR_OUTPUT
    OutSpeed : INT;  (* Speed Setting *)
    OutAcc : UINT;  (* Acc Setting *)
    OutDec : UINT;  (* Dec Setting *)
    ControlWord : UINT;
END_VAR
VAR_EXTERNAL
    ResetAlarmes : BOOL;
END_VAR
VAR
    _p1 : BOOL;
END_VAR
(* ladder, written here as Structured Text *)

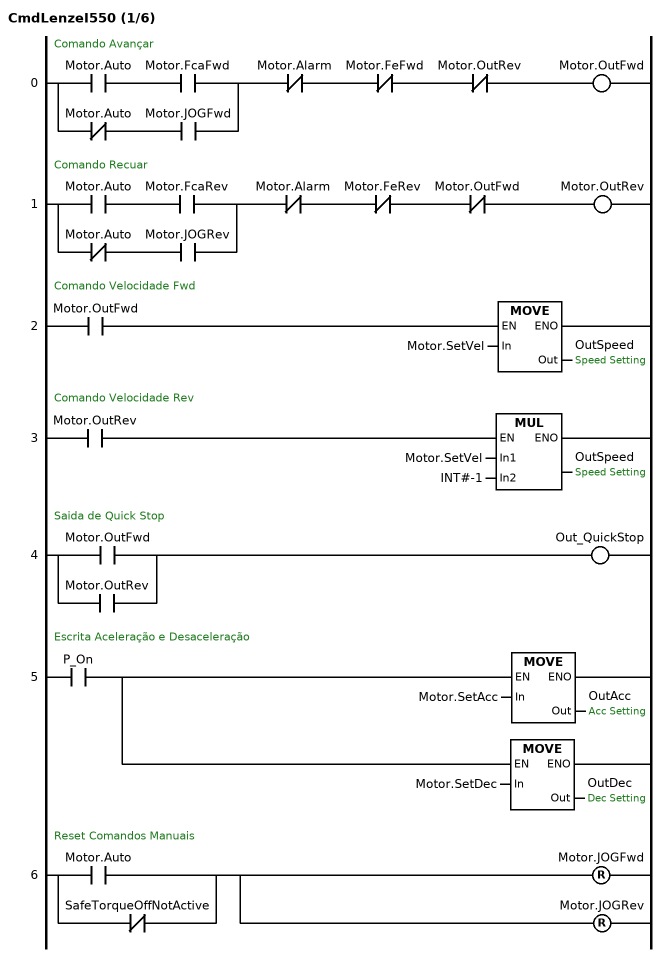
(* Rung 0: Comando Avançar *)
Motor.OutFwd := ((Motor.Auto AND Motor.FcaFwd) OR (NOT Motor.Auto AND Motor.JOGFwd)) AND NOT Motor.Alarm AND NOT Motor.FeFwd AND NOT Motor.OutRev;
(* Rung 1: Comando Recuar *)
Motor.OutRev := ((Motor.Auto AND Motor.FcaRev) OR (NOT Motor.Auto AND Motor.JOGRev)) AND NOT Motor.Alarm AND NOT Motor.FeRev AND NOT Motor.OutFwd;
(* Rung 2: Comando Velocidade Fwd *)
IF Motor.OutFwd THEN OutSpeed := Motor.SetVel; END_IF;
(* Rung 3: Comando Velocidade Rev *)
IF Motor.OutRev THEN OutSpeed := Motor.SetVel * (INT#-1); END_IF;
(* Rung 4: Saida de Quick Stop *)
Out_QuickStop := Motor.OutFwd OR Motor.OutRev;
(* Rung 5: Escrita Aceleração e Desaceleração *)
IF P_On THEN
    OutAcc := Motor.SetAcc;
    OutDec := Motor.SetDec;
END_IF;
(* Rung 6: Reset Comandos Manuais *)
_p1 := Motor.Auto OR NOT SafeTorqueOffNotActive;
IF _p1 THEN
    Motor.JOGFwd := FALSE;
    Motor.JOGRev := FALSE;
END_IF;

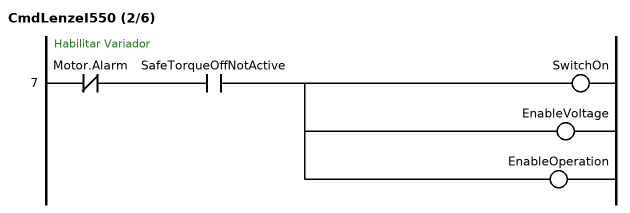
(* Rung 7: Habilitar Variador *)
SwitchOn := NOT Motor.Alarm AND SafeTorqueOffNotActive;
EnableVoltage := NOT Motor.Alarm AND SafeTorqueOffNotActive;
EnableOperation := NOT Motor.Alarm AND SafeTorqueOffNotActive;

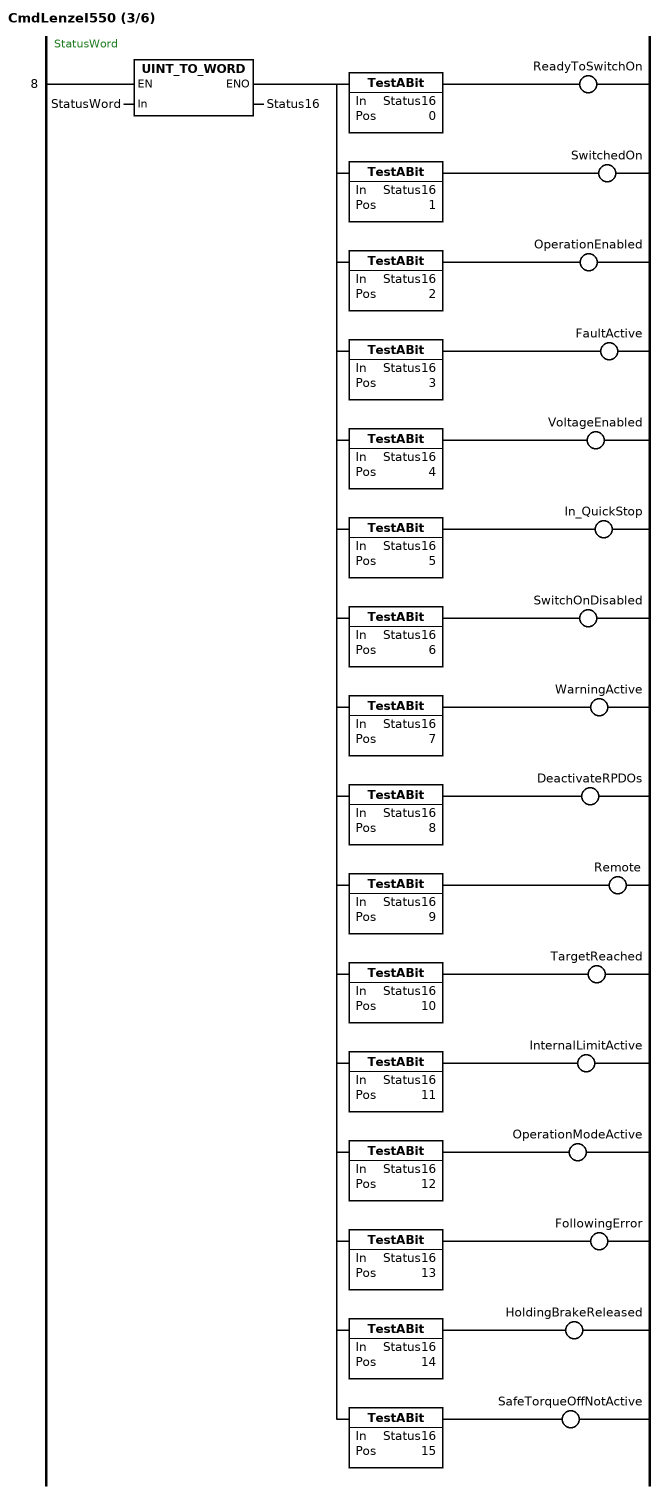
(* Rung 8: StatusWord *)
Status16 := UINT_TO_WORD(In := StatusWord);
ReadyToSwitchOn := TestABit(In := Status16, Pos := 0);
SwitchedOn := TestABit(In := Status16, Pos := 1);
OperationEnabled := TestABit(In := Status16, Pos := 2);
FaultActive := TestABit(In := Status16, Pos := 3);
VoltageEnabled := TestABit(In := Status16, Pos := 4);
In_QuickStop := TestABit(In := Status16, Pos := 5);
SwitchOnDisabled := TestABit(In := Status16, Pos := 6);
WarningActive := TestABit(In := Status16, Pos := 7);
DeactivateRPDOs := TestABit(In := Status16, Pos := 8);
Remote := TestABit(In := Status16, Pos := 9);
TargetReached := TestABit(In := Status16, Pos := 10);
InternalLimitActive := TestABit(In := Status16, Pos := 11);
OperationModeActive := TestABit(In := Status16, Pos := 12);
FollowingError := TestABit(In := Status16, Pos := 13);
HoldingBrakeReleased := TestABit(In := Status16, Pos := 14);
SafeTorqueOffNotActive := TestABit(In := Status16, Pos := 15);

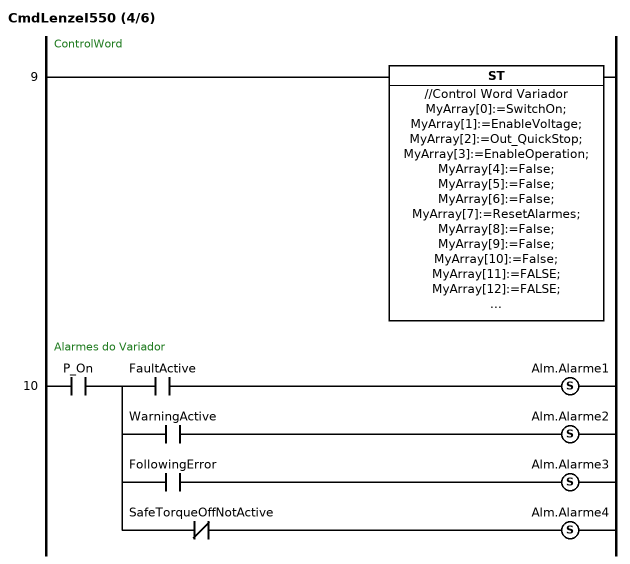
(* Rung 9: ControlWord *)
//Control Word Variador

MyArray[0]:=SwitchOn;
MyArray[1]:=EnableVoltage;
MyArray[2]:=Out_QuickStop;
MyArray[3]:=EnableOperation;
MyArray[4]:=False;
MyArray[5]:=False;
MyArray[6]:=False;
MyArray[7]:=ResetAlarmes;
MyArray[8]:=False;
MyArray[9]:=False;
MyArray[10]:=False;
MyArray[11]:=FALSE;
MyArray[12]:=FALSE;
MyArray[13]:=False;
MyArray[14]:=FALSE;
MyArray[15]:=False;
ControlWord:=BitArray16_to_UInt(MyArray);
(* Rung 10: Alarmes do Variador *)
IF P_On AND FaultActive THEN Alm.Alarme1 := TRUE; END_IF;
IF P_On AND WarningActive THEN Alm.Alarme2 := TRUE; END_IF;
IF P_On AND FollowingError THEN Alm.Alarme3 := TRUE; END_IF;
IF P_On AND NOT SafeTorqueOffNotActive THEN Alm.Alarme4 := TRUE; END_IF;

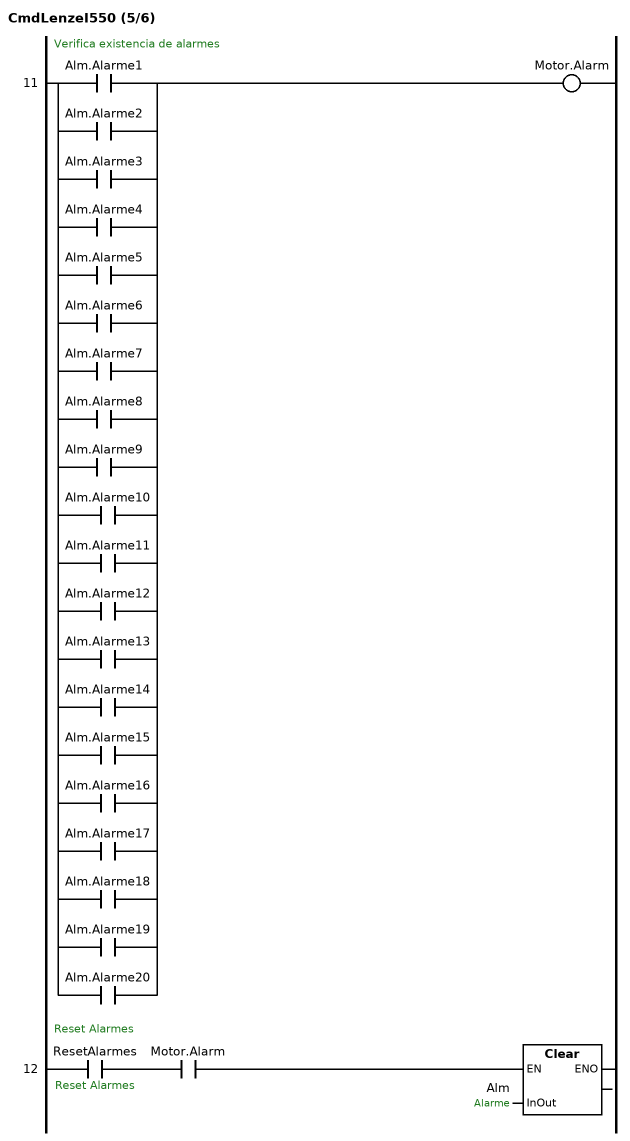
(* Rung 11: Verifica existencia de alarmes *)
Motor.Alarm := Alm.Alarme1 OR Alm.Alarme2 OR Alm.Alarme3 OR Alm.Alarme4 OR Alm.Alarme5 OR Alm.Alarme6 OR Alm.Alarme7 OR Alm.Alarme8 OR Alm.Alarme9 OR Alm.Alarme10 OR Alm.Alarme11 OR Alm.Alarme12 OR Alm.Alarme13 OR Alm.Alarme14 OR Alm.Alarme15 OR Alm.Alarme16 OR Alm.Alarme17 OR Alm.Alarme18 OR Alm.Alarme19 OR Alm.Alarme20;
(* Rung 12: Reset Alarmes *)
IF ResetAlarmes AND Motor.Alarm THEN Clear(InOut := Alm); END_IF;

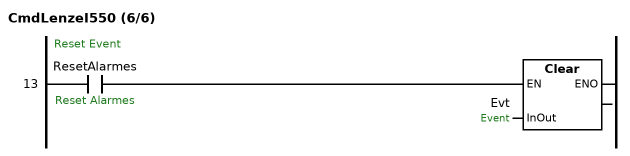
(* Rung 13: Reset Event *)
IF ResetAlarmes THEN Clear(InOut := Evt); END_IF;
END_FUNCTION_BLOCK

FUNCTION_BLOCK CmdMotor
VAR_INPUT
    Enable : BOOL;
END_VAR
VAR_IN_OUT
    Motor : DataMotor;  (* Data *)
    Alm : AlarmeGeralEquipamento;  (* Alarme *)
    Evt : Event;  (* Event *)
END_VAR
VAR_EXTERNAL
    ResetAlarmes : BOOL;
END_VAR
VAR
    _p1 : BOOL;
END_VAR
(* ladder, written here as Structured Text *)

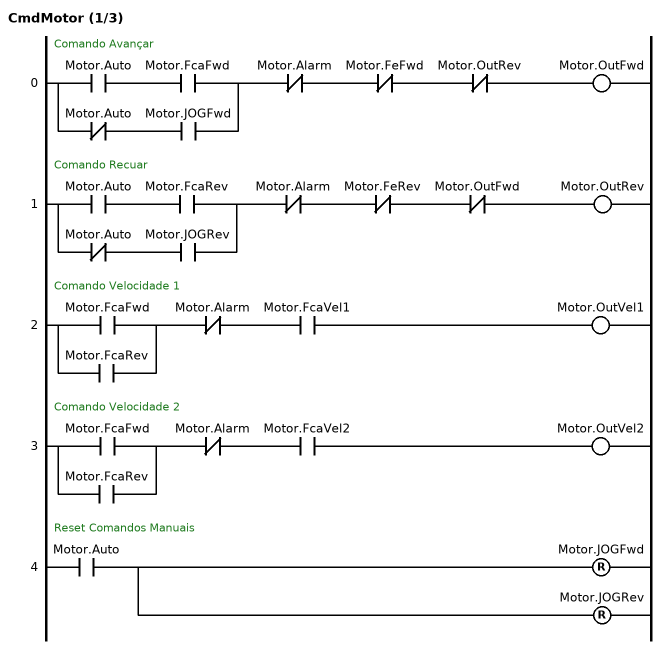
(* Rung 0: Comando Avançar *)
Motor.OutFwd := ((Motor.Auto AND Motor.FcaFwd) OR (NOT Motor.Auto AND Motor.JOGFwd)) AND NOT Motor.Alarm AND NOT Motor.FeFwd AND NOT Motor.OutRev;
(* Rung 1: Comando Recuar *)
Motor.OutRev := ((Motor.Auto AND Motor.FcaRev) OR (NOT Motor.Auto AND Motor.JOGRev)) AND NOT Motor.Alarm AND NOT Motor.FeRev AND NOT Motor.OutFwd;
(* Rung 2: Comando Velocidade 1 *)
Motor.OutVel1 := (Motor.FcaFwd OR Motor.FcaRev) AND NOT Motor.Alarm AND Motor.FcaVel1;
(* Rung 3: Comando Velocidade 2 *)
Motor.OutVel2 := (Motor.FcaFwd OR Motor.FcaRev) AND NOT Motor.Alarm AND Motor.FcaVel2;
(* Rung 4: Reset Comandos Manuais *)
_p1 := Motor.Auto;
IF _p1 THEN
    Motor.JOGFwd := FALSE;
    Motor.JOGRev := FALSE;
END_IF;

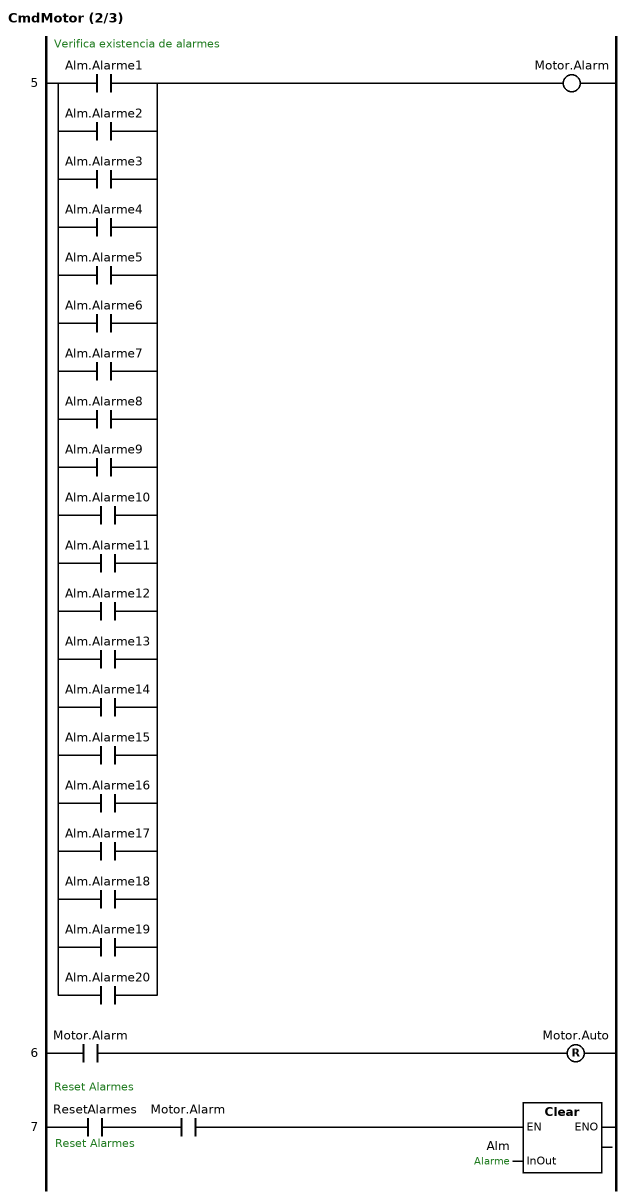
(* Rung 5: Verifica existencia de alarmes *)
Motor.Alarm := Alm.Alarme1 OR Alm.Alarme2 OR Alm.Alarme3 OR Alm.Alarme4 OR Alm.Alarme5 OR Alm.Alarme6 OR Alm.Alarme7 OR Alm.Alarme8 OR Alm.Alarme9 OR Alm.Alarme10 OR Alm.Alarme11 OR Alm.Alarme12 OR Alm.Alarme13 OR Alm.Alarme14 OR Alm.Alarme15 OR Alm.Alarme16 OR Alm.Alarme17 OR Alm.Alarme18 OR Alm.Alarme19 OR Alm.Alarme20;
(* Rung 6 *)
IF Motor.Alarm THEN Motor.Auto := FALSE; END_IF;
(* Rung 7: Reset Alarmes *)
IF ResetAlarmes AND Motor.Alarm THEN Clear(InOut := Alm); END_IF;

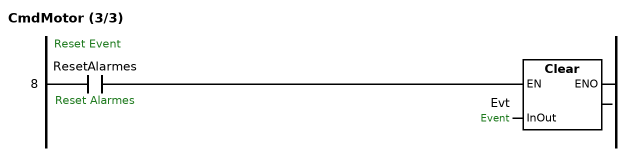
(* Rung 8: Reset Event *)
IF ResetAlarmes THEN Clear(InOut := Evt); END_IF;
END_FUNCTION_BLOCK

FUNCTION_BLOCK CmdValve
VAR_IN_OUT
    Valve : DataValve;  (* Data *)
    Alm : AlarmeGeralEquipamento;  (* Alarme *)
    Evt : Event;  (* Event *)
END_VAR
VAR_INPUT
    Enable : BOOL;
END_VAR
VAR_EXTERNAL
    ResetAlarmes : BOOL;
END_VAR
VAR
    _p1 : BOOL;
END_VAR
(* ladder, written here as Structured Text *)

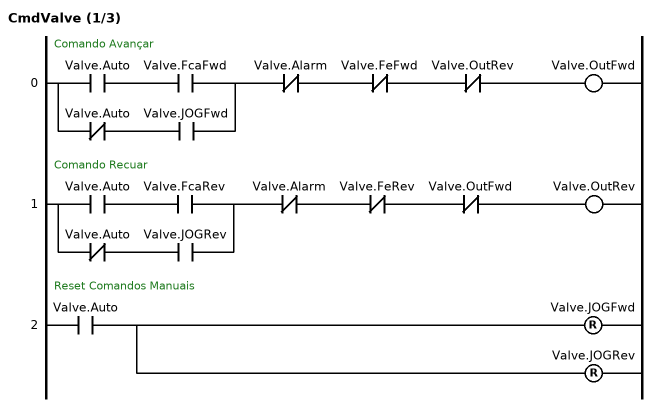
(* Rung 0: Comando Avançar *)
Valve.OutFwd := ((Valve.Auto AND Valve.FcaFwd) OR (NOT Valve.Auto AND Valve.JOGFwd)) AND NOT Valve.Alarm AND NOT Valve.FeFwd AND NOT Valve.OutRev;
(* Rung 1: Comando Recuar *)
Valve.OutRev := ((Valve.Auto AND Valve.FcaRev) OR (NOT Valve.Auto AND Valve.JOGRev)) AND NOT Valve.Alarm AND NOT Valve.FeRev AND NOT Valve.OutFwd;
(* Rung 2: Reset Comandos Manuais *)
_p1 := Valve.Auto;
IF _p1 THEN
    Valve.JOGFwd := FALSE;
    Valve.JOGRev := FALSE;
END_IF;

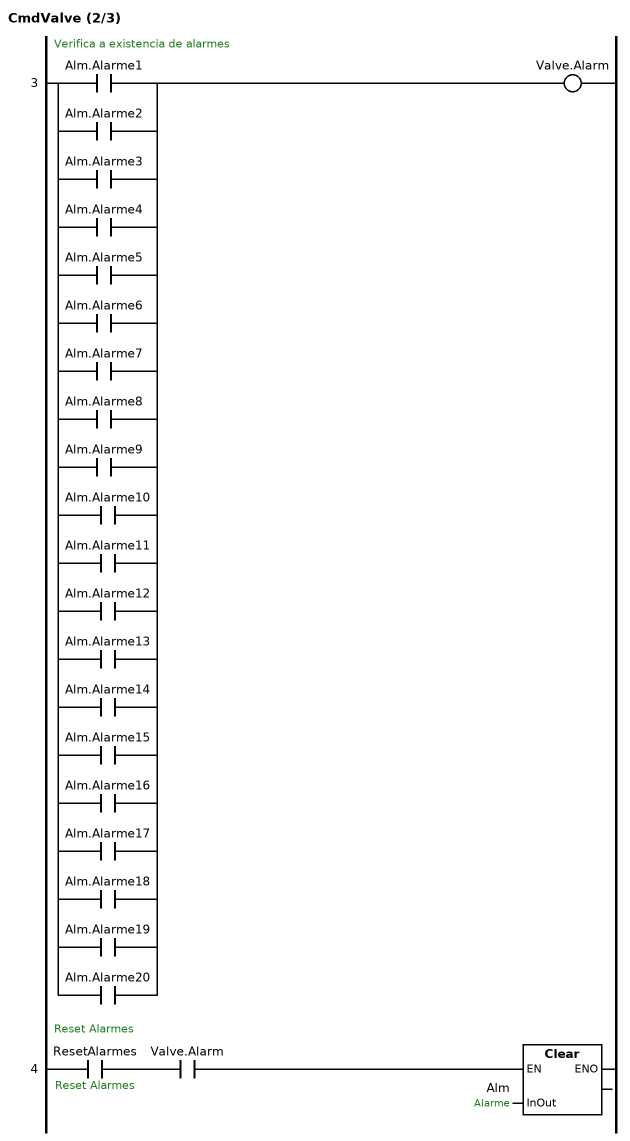
(* Rung 3: Verifica a existencia de alarmes *)
Valve.Alarm := Alm.Alarme1 OR Alm.Alarme2 OR Alm.Alarme3 OR Alm.Alarme4 OR Alm.Alarme5 OR Alm.Alarme6 OR Alm.Alarme7 OR Alm.Alarme8 OR Alm.Alarme9 OR Alm.Alarme10 OR Alm.Alarme11 OR Alm.Alarme12 OR Alm.Alarme13 OR Alm.Alarme14 OR Alm.Alarme15 OR Alm.Alarme16 OR Alm.Alarme17 OR Alm.Alarme18 OR Alm.Alarme19 OR Alm.Alarme20;
(* Rung 4: Reset Alarmes *)
IF ResetAlarmes AND Valve.Alarm THEN Clear(InOut := Alm); END_IF;

